TYPE ST_DALI102Parameters :
STRUCT
	nShortAddress			:	BYTE;	// 255: no short address
	nActualLevel			:	BYTE;
	nMinLevel				:	BYTE;
	nMaxLevel				: 	BYTE;
	eFadeRate				:	E_DALIFadeRate;
	eFadeTime				:	E_DALIFadeTime;
	nPowerOnLevel			:	BYTE;
	nSystemFailureLevel		:	BYTE;
	nPhysicalMinimum		:	BYTE;
	sDeviceTypes			:	STRING[100];
END_STRUCT
END_TYPE

(* stored: Version 1.1.0.1
   DUT ST_DALI102Parameters: Id {b2ce86f1-dd21-4bc2-8fc0-1b833db41f95} *)
